PROGRAM PrgMqttCom
VAR
	
	StartMosquitto : BOOL :=FALSE;
	fbMosquittoLaunch: NT_StartProcess;
	
	fbMqttClient : FB_IotMqttClient;
	bSetParameter : BOOL := TRUE ;
	bConnect : BOOL := TRUE ;
	
	(* published message *)
	sTopicPub : STRING(255) := 'remote/thingspeak/1226961/publish/H1SCE16XLESMI7KP'; //channelID and writeAPIkey must be changed to your own
	// from thingspeak channel profile
	sPayloadPub : STRING(255);
	i: UDINT := 0 ;
	switch : BOOL := TRUE;
	fbTimer : TON := (PT:=T#15S);
	
	(* received message *)
	(*bSubscribed : BOOL;
	sTopicSub : STRING(255) := 'test';
	{attribute 'TcEncoding':='UTF-8'}
	sTopicRcv : STRING(255);
	{attribute 'TcEncoding':='UTF-8'}
	sPayloadRcv : STRING(255);
	fbMessageQueue : FB_IotMqttMessageQueue;
	fbMessage : FB_IotMqttMessage;*)
	
	hrErrorOccurred : HRESULT; // contains the latest occurred error
	TMOUT: TIME;
	partAtSensor: BOOL;
	partCount: INT;
END_VAR

IF bSetParameter THEN
	fbMqttClient.sHostName:= '192.168.43.246'; // address of host, your computer and adpter
	fbMqttClient.nHostPort:= 1883; // port which bridge are listening to
	fbMqttClient.sTopicPrefix:= ''; 
	bSetParameter := FALSE;
END_IF

// This is for starting mosquitto, you can modify this or then just start mosquitto manually
//IF StartMosquitto THEN
//	fbMosquittoLaunch( PATHSTR :='c:\Program Files (x86)\mosquitto\Mosquitto.exe',
//					  COMNDLINE:='-c E:\AFOF\IOTTask\mosquittoConfFiles\thingSpeakBridgeTLS.conf'	,
//						START :=  StartMosquitto, 
//						TMOUT := T#3S);
						
	//StartMosquitto :=FALSE;
//END_IF

(*establishing cnnection*)
fbMqttClient.Execute(bConnect);
IF fbMqttClient.bError THEN
	// add your error logging here
	hrErrorOccurred := fbMqttClient.hrErrorCode;
END_IF

(* get messages from subscribed topic *)
(*IF fbMessageQueue.nQueuedMessages > 0 THEN
	IF fbMessageQueue.Dequeue(fbMessage:=fbMessage) THEN
		fbMessage.GetTopic(pTopic:=ADR(sTopicRcv), nTopicSize:=SIZEOF(sTopicRcv) );
		fbMessage.GetPayload(pPayload:=ADR(sPayloadRcv), nPayloadSize:=SIZEOF(sPayloadRcv), bSetNullTermination:=FALSE);
	END_IF
END_IF*)

IF fbMqttClient.bConnected THEN
	(* Subscribe to topuc *)
	(*IF NOT bSubscribed THEN
		bSubscribed := fbMqttClient.Subscribe(sTopic:=sTopicSub, eQoS:=TcIotMqttQos.AtMostOnceDelivery);
		IF fbMqttClient.bError THEN
			// add your error logging here
			hrErrorOccurred := fbMqttClient.hrErrorCode;
		END_IF
	END_IF*)
	fbTimer(IN:=TRUE);
	//IF fbTimer.Q THEN // publish new payload every 15 second
		//fbTimer(IN:=FALSE);
		IF partAtSensor THEN
			partCount := partCount + 1;
			partAtSensor := FALSE;
		END_IF
		fbMqttClient.Publish(	sTopic:= sTopicPub, 
								pPayload:= ADR(sPayloadPub), nPayloadSize:= LEN2(ADR(sPayloadPub))+1, 
								eQoS:= TcIotMqttQos.AtMostOnceDelivery, bRetain:= FALSE, bQueue:= FALSE );
								sPayloadPub := CONCAT('field1=', TO_STRING(partCount));
		IF fbMqttClient.bError THEN
			// add your error logging here
			hrErrorOccurred := fbMqttClient.hrErrorCode;
		END_IF
	END_IF
//END_IF

END_PROGRAM

(* stored: Version 1.1.0.1, ProductVersion 3.1.4024.5
   POU PrgMqttCom: Id {c70f107a-6ca5-4bfb-b775-e2929cbf9dae}, SpecialFunc None *)
